// TIA Portal V17 export
// export: Created 2025-04-09T08:03:58.8280717Z, ExportSetting WithDefaults, DisplayName Totally Integrated Automation Portal, DisplayVersion V17 Update 8, DisplayName TIA Portal Openness, DisplayVersion V17 Update 8, DisplayName TIA Portal Version Control Interface, DisplayVersion V17, DisplayName SINAMICS Startdrive Advanced, DisplayVersion V17 SP2, DisplayName SINAMICS Startdrive G110M, G120, G120C, G120D, G120P, G115D, DisplayVersion V17 SP2, DisplayName SINAMICS Startdrive G130, G150, S120, S150, SINAMICS MV, S210, DisplayVersion V17 SP2, DisplayName STEP 7 Professional, DisplayVersion V17 Update 8, DisplayName SINUMERIK ONE STEP 7 Toolbox, DisplayVersion V17 Update 12, DisplayName SINUMERIK ONE PLC Basic Program Plus, DisplayVersion V17 Update 12, DisplayName SINUMERIK 840D sl STEP 7 Toolbox, DisplayVersion V17 Update 12, DisplayName STEP 7 Safety, DisplayVersion V17 Update 6, DisplayName WinCC Advanced, DisplayVersion V17 Update 8
DATA_BLOCK "DB1201_PART_CYCLE_UNIT_1"   // DB1201
{ S7_Optimized_Access := 'FALSE'; DB_Accessible_From_OPC_UA := 'FALSE' }
AUTHOR : ETXETAR
VERSION : 1.0
// stored: AutoNumber false, DBAccessibleFromOPCUA false, DBAccessibleFromWebserver true, IsOnlyStoredInLoadMemory false, IsWriteProtectedInAS false
   VAR RETAIN
      GENERAL_CONDITIONS : Bool;   // GENERAL CONDITIONS
      INITIAL_CONDITIONS : Bool;   // INITIAL CONDITIONS
      REQUEST : Bool;   // REQUEST
      REQUEST_PULSE : Bool;   // REQUEST PULSE
      COMMAND : Bool;   // COMMAND
      COMMAND_PULSE : Bool;   // COMMAND PULSE
      RUNNING : Bool;   // RUNNING
      SPARE : Bool;
      CYCLE_UNIT_01_STATION_0 : Bool;   // CYCLE UNIT 01 STATION 0 START REQUEST
      CYCLE_UNIT_01_STATION_1 : Bool;   // CYCLE UNIT 01 STATION 1 START REQUEST
      CYCLE_UNIT_01_STATION_2 : Bool;   // CYCLE UNIT 01 STATION 2 START REQUEST
      CYCLE_UNIT_01_STATION_3 : Bool;   // CYCLE UNIT 01 STATION 3 START REQUEST
      CYCLE_UNIT_01_STATION_4 : Bool;   // CYCLE UNIT 01 STATION 4 START REQUEST
      UNIT_01_CALIBRATION_STATION_3 : Bool;   // UNIT 01 STATION 3 MASTER CALIBRATION CYCLE REQUEST
      UNIT_01_MASTER_MEASUREMENT_STATION_3 : Bool;   // UNIT 01 STATION 3 MASTER MEASUREMENT CYCLE REQUEST
      U01_STA_1_COND_OK_STA_0_CYCLE : Bool;   // UNIT 01 STATION 1 CONDITIONS OK FOR STATION 0 CYCLE REQUEST
      U01_STA_2_COND_OK_STA_0_CYCLE : Bool;   // UNIT 01 STATION 2 CONDITIONS OK FOR STATION 0 CYCLE REQUEST
      U01_STA_3_COND_OK_STA_0_CYCLE : Bool;   // UNIT 01 STATION 3 CONDITIONS OK FOR STATION 0 CYCLE REQUEST
      U01_STA_4_COND_OK_STA_0_CYCLE : Bool;   // UNIT 01 STATION 4 CONDITIONS OK FOR STATION 0 CYCLE REQUEST
      U01_NEW_FACE_STA_1 : Bool;   // UNIT 01 NEW FACE IN STATION 1
      U01_FACE_DONE_STA_1 : Bool;   // UNIT 01 FACE DONE IN STATION 1
      RESET_PLC_AND_CNC : Bool;   // RESET PLC AND CNC
      HMI_SEMI_REQUEST : Bool;   // HMI PUSHBUTTON SEMI REQUEST
      SEMI_AUTO_REQUEST : Bool;   // SEMI AUTO REQUEST
      SEMI_AUTO_REQUEST_PULSE : Bool;   // SEMI AUTO REQUEST PULSE
      AUTO_REQUEST : Bool;   // AUTO REQUEST
      FULL_DEPTH : Bool;   // FULL DEPTH
      TIME_EXCEEDED : Bool;   // TIME EXCEEDED ALARM
      PREALARM : Bool;   // PREALARM
      AUX0 : Bool;   // AUXILIARY 0
      AUX1 : Bool;   // AUXILIARY 1
      AUX2 : Bool;   // AUXILIARY 2
      AUX3 : Bool;   // AUXILIARY 3
      AUX5 : Bool;   // AUXILIARY 5
      AUX6 : Bool;   // AUXILIARY 6
      AUX7 : Bool;   // AUXILIARY 7
      PREALARM_GONE : Bool;   // PREALARM GONE
      GENERAL_CONDITIONS_HELP : Bool;   // GENERAL CONDITIONS HELP
      INITIAL_CONDITIONS_HELP : Bool;   // INITIAL CONDITIONS HELP
      TIMER_TIME_EXCEED : TON_TIME;   // TIME EXCEEDED TIMER
      SEQUENCE : "RUN_CNC_SEQ";
   END_VAR
BEGIN
   TIMER_TIME_EXCEED.PT := T#800s;
   SEQUENCE.TIMER_TIME_EXCEED.PT := T#500s;
END_DATA_BLOCK
